# B&R Automation Studio project NAEUL004C00R13L518F00 (part 43)

#### Local.var
```iecst
(*2019-10-30*)
(**)
(*Local Action, State & Status*)
VAR
	eAct : eMagConv2ClpAction := MagConv2ClpActIdle;
	eStat : eMagConv2ClpAction := MagConv2ClpActIdle;
	eStatus : eFBStatus := Idle;
	udiStatus : UDINT := 0;
	sStatTxt : STRING[200] := '';
	a_sStatText : ARRAY[0..50] OF STRING[200] := ['Idling','Initializing','Initializing With Stop Then Clamper','Initializing With Clamper Then Stop','Entering Board','Entering Board With Stop Then Clamper','Entering Board With Clamper Then Stop','Pre-Exiting Board','Pre-Exiting Board With Clamper',2('Exiting Board'),2('Exiting Board With Clamper'),'Fix/Bottom Clamper Setting All Control','Fix/Bottom Clamper Resetting All Control','Fix/Bottom Clamper Setting Clamp','Fix/Bottom Clamper Setting Unclamp','Fix/Bottom Clamper Clamp','Fix/Bottom Clampler Unclamp','Remote/Top Clamper Setting All Control','Remote/Top Clamper Resetting All Control','Remote/Top Clamper Setting Clamp','Remote/Top Clamper Setting Unclamp','Remote/Top Clamper Clamp','Remote/Top Clampler Unclamp','Stopping','Stopping With Clamper','Turning On Motor Signal','Turning On Motor Direction','Turning Off Motor Signal','Turning Off Motor Direction','Turning On All Motor Output','Turning Off All Motor Output',18('')];
END_VAR
(**)
(*Local Alarm*)
VAR
	tyAlmData : tyAlmDat;
	a_tyAlmText : ARRAY[10000..10099] OF tyAlmTxt := [(sAlmText:='Magazine Detected But Not Present At Outlet Sensor (L - R) While Magazine Conveyor Initial',sRcyText:='Operation Interrupted By Undetected Magazine. Adjusting The Magazine Or Remove The Present Magazine To Resume Operation.'),(sAlmText:='Magazine Detected But Not Present At Outlet Sensor (R - L) While Magazine Conveyor Initial',sRcyText:='Operation Interrupted By Undetected Magazine. Adjusting The Magazine Or Remove The Present Magazine To Resume Operation.'),(sAlmText:='Clamper Clamp Sensor Off Time Out In Unclamp Check While Conveyor Initial With Clamper',sRcyText:='Sensor Timeout Expired Before Operation Completed. Sensor Operation Is Abnormal. Solve The Error To Resume Operation.'),(sAlmText:='Clamper Unclamp Sensor On Time Out In Unclamp Check While Conveyor Initial With Clamper',sRcyText:='Sensor Timeout Expired Before Operation Completed. Sensor Operation Is Abnormal. Solve The Error To Resume Operation.'),(sAlmText:='Clamper Unclamp Safety Sensor Error In Unclamp Check While Conveyor Initial With Clamper',sRcyText:='Safety System Has Been Triggered. All Operations Are Disable. Remove the Obstacle That Triggered The Safety Interlock To Resume Operation.'),(sAlmText:='Magazine Detected But Not Present At Outlet Sensor (L - R) While Conveyor Initial With Clamper',sRcyText:='Operation Interrupted By Undetected Magazine. Adjusting The Magazine Or Remove The Present Magazine To Resume Operation.'),(sAlmText:='Magazine Detected But Not Present At Outlet Sensor (R - L) While Conveyor Initial With Clamper',sRcyText:='Operation Interrupted By Undetected Magazine. Adjusting The Magazine Or Remove The Present Magazine To Resume Operation.'),(sAlmText:='Clamper Clamp Sensor On Time Out In Clamp Check While Conveyor Initial With Clamper',sRcyText:='Sensor Timeout Expired Before Operation Completed. Sensor Operation Is Abnormal. Solve The Error To Resume Operation.'),(sAlmText:='Clamper Unclamp Sensor Off Time Out In Clamp Check While Conveyor Initial With Clamper',sRcyText:='Sensor Timeout Expired Before Operation Completed. Sensor Operation Is Abnormal. Solve The Error To Resume Operation.'),(sAlmText:='Clamper Clamp Safety Sensor Error In Clamp Check While Conveyor Initial With Clamper',sRcyText:='Safety System Has Been Triggered. All Operations Are Disable. Remove the Obstacle That Triggered The Safety Interlock To Resume Operation.'),(sAlmText:='Clamper Clamp Sensor On Time Out In Clamp Check While Conveyor Enter With Clamper',sRcyText:='Sensor Timeout Expired Before Operation Completed. Sensor Operation Is Abnormal. Solve The Error To Resume Operation.'),(sAlmText:='Clamper Unclamp Sensor Off Time Out In Clamp Check While Conveyor Enter With Clamper',sRcyText:='Sensor Timeout Expired Before Operation Completed. Sensor Operation Is Abnormal. Solve The Error To Resume Operation.'),(sAlmText:='Clamper Clamp Safety Sensor Error In Clamp Check While Conveyor Enter With Clamper',sRcyText:='Safety System Has Been Triggered. All Operations Are Disable. Remove the Obstacle That Triggered The Safety Interlock To Resume Operation.'),(sAlmText:='Clamper Clamp Sensor Off Time Out In Unclamp Check While Conveyor Exit With Clamper',sRcyText:='Sensor Timeout Expired Before Operation Completed. Sensor Operation Is Abnormal. Solve The Error To Resume Operation.'),(sAlmText:='Clamper Unclamp Sensor On Time Out In Unclamp Check While Conveyor Exit With Clamper',sRcyText:='Sensor Timeout Expired Before Operation Completed. Sensor Operation Is Abnormal. Solve The Error To Resume Operation.'),(sAlmText:='Clamper Unclamp Safety Sensor Error In Unclamp Check While Conveyor Exit With Clamper',sRcyText:='Safety System Has Been Triggered. All Operations Are Disable. Remove the Obstacle That Triggered The Safety Interlock To Resume Operation.'),(sAlmText:='Clamper Clamp Sensor On Time Out In Clamp Check While Clamper Clamp',sRcyText:='Sensor Timeout Expired Before Operation Completed. Sensor Operation Is Abnormal. Solve The Error To Resume Operation.'),(sAlmText:='Clamper Unclamp Sensor Off Time Out In Clamp Check While Clamper Clamp',sRcyText:='Sensor Timeout Expired Before Operation Completed. Sensor Operation Is Abnormal. Solve The Error To Resume Operation.'),(sAlmText:='Clamper Clamp Safety Sensor Error In Clamp Check While Clamper Clamp',sRcyText:='Safety System Has Been Triggered. All Operations Are Disable. Remove the Obstacle That Triggered The Safety Interlock To Resume Operation.'),(sAlmText:='Clamper Clamp Sensor Off Time Out In Unclamp Check While Clamper Unclamp',sRcyText:='Sensor Timeout Expired Before Operation Completed. Sensor Operation Is Abnormal. Solve The Error To Resume Operation.'),(sAlmText:='Clamper Unclamp Sensor On Time Out In Unclamp Check While Clamper Unclamp',sRcyText:='Sensor Timeout Expired Before Operation Completed. Sensor Operation Is Abnormal. Solve The Error To Resume Operation.'),(sAlmText:='Clamper Unclamp Safety Sensor Error In Unclamp Check While Clamper Unclamp',sRcyText:='Safety System Has Been Triggered. All Operations Are Disable. Remove the Obstacle That Triggered The Safety Interlock To Resume Operation.'),(sAlmText:='Clamper Clamp Sensor Off Time Out In Unclamp Check While Stop With Clamper',sRcyText:='Sensor Timeout Expired Before Operation Completed. Sensor Operation Is Abnormal. Solve The Error To Resume Operation.'),(sAlmText:='Clamper Unclamp Sensor On Time Out In Unclamp Check While Stop With Clamper',sRcyText:='Sensor Timeout Expired Before Operation Completed. Sensor Operation Is Abnormal. Solve The Error To Resume Operation.'),(sAlmText:='Clamper Unclamp Safety Sensor Error In Unclamp Check While Stop With Clamper',sRcyText:='Safety System Has Been Triggered. All Operations Are Disable. Remove the Obstacle That Triggered The Safety Interlock To Resume Operation.'),(sAlmText:='Clamper Clamp Sensor Off Time Out In Unclamp Check While Conveyor Exit With Clamper',sRcyText:='Sensor Timeout Expired Before Operation Completed. Sensor Operation Is Abnormal. Solve The Error To Resume Operation.'),(sAlmText:='Clamper Unclamp Sensor On Time Out In Unclamp Check While Conveyor Exit With Clamper',sRcyText:='Sensor Timeout Expired Before Operation Completed. Sensor Operation Is Abnormal. Solve The Error To Resume Operation.'),(sAlmText:='Clamper Unclamp Safety Sensor Error In Unclamp Check While Conveyor Exit With Clamper',sRcyText:='Safety System Has Been Triggered. All Operations Are Disable. Remove the Obstacle That Triggered The Safety Interlock To Resume Operation.'),2((sAlmText:='Transfer In Time Out While Entering Magazine',sRcyText:='Timeout Expired Before Operation Completed. Transmission Abnormal. Remove the Obstacle (If Exists) To Resume Operation.')),(sAlmText:='Transfer Out Time Out While Exiting Magazine',sRcyText:='Timeout Expired Before Operation Completed. Transmission Abnormal. Remove the Obstacle (If Exists) To Resume Operation.'),(sAlmText:='Transfer Out Time Out While Conveyor Exit With Clamper',sRcyText:='Timeout Expired Before Operation Completed. Transmission Abnormal. Remove the Obstacle (If Exists) To Resume Operation.'),(sAlmText:='Transfer Out Time Out While Exiting Magazine',sRcyText:='Timeout Expired Before Operation Completed. Transmission Abnormal. Remove the Obstacle (If Exists) To Resume Operation.'),(sAlmText:='Transfer Out Time Out While Conveyor Exit With Clamper',sRcyText:='Timeout Expired Before Operation Completed. Transmission Abnormal. Remove the Obstacle (If Exists) To Resume Operation.'),(sAlmText:='Clamper Clamp Sensor On Time Out In Clamp Check While Conveyor Enter With Clamper',sRcyText:='Sensor Timeout Expired Before Operation Completed. Sensor Operation Is Abnormal. Solve The Error To Resume Operation.'),(sAlmText:='Clamper Unclamp Sensor Off Time Out In Clamp Check While Conveyor Enter With Clamper',sRcyText:='Sensor Timeout Expired Before Operation Completed. Sensor Operation Is Abnormal. Solve The Error To Resume Operation.'),(sAlmText:='Clamper Clamp Safety Sensor Error In Clamp Check While Conveyor Enter With Clamper',sRcyText:='Safety System Has Been Triggered. All Operations Are Disable. Remove the Obstacle That Triggered The Safety Interlock To Resume Operation.'),(sAlmText:='Transfer In Time Out While Entering Magazine',sRcyText:='Timeout Expired Before Operation Completed. Transmission Abnormal. Remove the Obstacle (If Exists) To Resume Operation.'),(sAlmText:='Clamper Clamp Sensor Off Time Out In Unclamp Check While Conveyor Initial With Clamper',sRcyText:='Sensor Timeout Expired Before Operation Completed. Sensor Operation Is Abnormal. Solve The Error To Resume Operation.'),(sAlmText:='Clamper Unclamp Sensor On Time Out In Unclamp Check While Conveyor Initial With Clamper',sRcyText:='Sensor Timeout Expired Before Operation Completed. Sensor Operation Is Abnormal. Solve The Error To Resume Operation.'),(sAlmText:='Clamper Unclamp Safety Sensor Error In Unclamp Check While Conveyor Initial With Clamper',sRcyText:='Safety System Has Been Triggered. All Operations Are Disable. Remove the Obstacle That Triggered The Safety Interlock To Resume Operation.'),(sAlmText:='Magazine Detected But Not Present At Outlet Sensor (L - R) While Conveyor Initial With Clamper',sRcyText:='Operation Interrupted By Undetected Magazine. Adjusting The Magazine Or Remove The Present Magazine To Resume Operation.'),(sAlmText:='Magazine Detected But Not Present At Outlet Sensor (R - L) While Conveyor Initial With Clamper',sRcyText:='Operation Interrupted By Undetected Magazine. Adjusting The Magazine Or Remove The Present Magazine To Resume Operation.'),(sAlmText:='Clamper Clamp Sensor On Time Out In Clamp Check While Conveyor Initial With Clamper',sRcyText:='Sensor Timeout Expired Before Operation Completed. Sensor Operation Is Abnormal. Solve The Error To Resume Operation.'),(sAlmText:='Clamper Unclamp Sensor Off Time Out In Clamp Check While Conveyor Initial With Clamper',sRcyText:='Sensor Timeout Expired Before Operation Completed. Sensor Operation Is Abnormal. Solve The Error To Resume Operation.'),(sAlmText:='Clamper Clamp Safety Sensor Error In Clamp Check While Conveyor Initial With Clamper',sRcyText:='Safety System Has Been Triggered. All Operations Are Disable. Remove the Obstacle That Triggered The Safety Interlock To Resume Operation.'),(sAlmText:='Magazine Not Detected While Pre-Exiting Magazine',sRcyText:='Operation Interrupted By Undetected Magazine. Adjusting The Magazine Or Remove The Present Magazine To Resume Operation.'),(sAlmText:='Magazine Width Check Sensor Deactivated',sRcyText:='Please Check the Magazine Width'),(sAlmText:='Saftey Sensor Is Deactivated To Clamp',sRcyText:='Please Check Safety Sensor'),51((0))];
END_VAR
(**)
(*Local Output*)
VAR
	bHvMag : BOOL := FALSE;
	bMtrSigOnOrLToR : BOOL := FALSE;
	bMtrDirOrRToL : BOOL := FALSE;
	bFixClprClampCtrl : BOOL;
	bRmtClprClampCtrl : BOOL;
	bClprTwoOutputControl : BOOL := FALSE;
END_VAR
(**)
(*Local Input*)
VAR
	udiRstErr : UDINT := 0;
	bPrep : BOOL := TRUE;
	bEn : BOOL := TRUE;
	bDis : BOOL := FALSE;
	bManual : BOOL := FALSE;
	bOnDirMod : BOOL := FALSE;
	diInitTm : DINT := 10000;
	tMtrOffDlyTm : TIME := T#0S;
	diTxInTimeOut : DINT := 10000;
	diTxOutTimeOut : DINT := 10000;
	eDirection : eConvDir := ConvDirLToR;
	bLeftSen : BOOL := FALSE;
	bRightSen : BOOL := FALSE;
	bFixClprClampSen : BOOL := FALSE;
	bFixClprUnclampSen : BOOL := FALSE;
	bFixClprClampSafetySen : BOOL := TRUE;
	bFixClprUnclampSafetySen : BOOL := TRUE;
	bRmtClprClampSen : BOOL := FALSE;
	bRmtClprUnclampSen : BOOL := FALSE;
	bRmtClprClampSafetySen : BOOL := TRUE;
	bRmtClprUnclampSafetySen : BOOL := TRUE;
	bWidthChkPrep : BOOL := TRUE;
	sProgNm : STRING[15] := 'MagConv2Clp';
	tClprClampTO : TIME := T#20s;
	tClprUnclampTO : TIME := T#20s;
	bNtSettingsLoadDone : BOOL := TRUE;
END_VAR
(**)
(*Local*)
VAR
	bRstErr : BOOL;
	udiRstErrOld : UDINT;
	bInitDone : BOOL;
	bInitialDone : BOOL;
	bReachEnd : BOOL;
	usiStep : USINT;
	usiSubStep : USINT;
	eStatOld : eMagConv2ClpAction := MagConv2ClpActIdle;
	fbInit : fbConvSenToSenTm;
	fbEnt : fbConvSenToSen;
	fbPreExit : fbConvSenToSenTm;
	fbExit : fbConvSenToSenOff;
	fbExit1 : fbConvSenToSenOff1;
	fbStop : fbConvMtrOff;
	fbFixClprClampChk : fbPneuExtRetSenExtChk;
	fbFixClprUnclampChk : fbPneuExtRetSenRetChk;
	fbRmtClprClampChk : fbPneuExtRetSenExtChk;
	fbFixClprDly : TON := (PT:=T#1s);
	fbRmtClprUnclampChk : fbPneuExtRetSenRetChk;
	fbClprDlyTm : TON;
	fbSmallLargeSenDlyTm : TON := (PT:=T#1S);
	fbWidthChk : TON := (PT:=T#30s);
	fbLeftSenDelayTm : TON := (PT:=T#1S);
	fbClpExtChkTm : TON := (PT:=T#200ms);
	udiModuleNum : UDINT := 1901;
END_VAR
```

#### Act_Alarm.st
```iecst
(** 2019-10-30 **)
ACTION Act_Alarm:
	//Reset Error
	IF (tylocalMagConv2Clp.Out.eStatus = Error) AND bRstErr THEN
		tylocalMagConv2Clp.In.eAct	:= MagConv2ClpActIdle;
		tylocalMagConv2Clp.Out.eStat	:= MagConv2ClpActIdle;
	END_IF

	IF tylocalMagConv2Clp.In.udiRstErr <> udiRstErrOld THEN
		bRstErr			:= TRUE;
		udiRstErrOld	:= tylocalMagConv2Clp.In.udiRstErr;
	ELSE
		bRstErr			:= FALSE;
	END_IF
	//Error
	IF EDGEPOS(tylocalMagConv2Clp.Out.eStatus = Error) THEN

		tylocalMagConv2Clp.Out.tyAlmData.sProgNm		:= tylocalMagConv2Clp.In.sProgNm;
		tylocalMagConv2Clp.Out.tyAlmData.udiCode		:= udiStatus;
		tylocalMagConv2Clp.Out.tyAlmData.eSeverity		:= AlmSeverityError;
		tylocalMagConv2Clp.Out.tyAlmData.udiRunTime	:= tylocalMagConv2Clp.Out.tyAlmData.udiRunTime + 1;
		tylocalMagConv2Clp.Out.tyAlmData.bAlm			:= TRUE;
		tylocalMagConv2Clp.Out.tyAlmData.udiModuleNum  := udiModuleNum;
		g_sMagConv2ClpProgNm		:= tylocalMagConv2Clp.In.sProgNm;
		tylocalMagConv2Clp.Out.sStatTxt	:= tylocalMagConv2Clp.Out.tyAlmData.sAlmMsg;

	ELSIF bRstErr AND (tylocalMagConv2Clp.Out.tyAlmData.udiCode <> 0) THEN

		tylocalMagConv2Clp.Out.tyAlmData.udiCode	:= 0;
		tylocalMagConv2Clp.Out.tyAlmData.eSeverity	:= AlmSeverityNA;
		tylocalMagConv2Clp.Out.tyAlmData.bAlm			:= FALSE;
		tylocalMagConv2Clp.Out.sStatTxt	:= a_sStatText[tylocalMagConv2Clp.Out.eStat];

	END_IF

END_ACTION
```

#### Act_InitGlobal.st
```iecst
(** 2019-10-30 **)
ACTION Act_InitGlobal:

	(* Always Change If Project Change *)

	//Pass Data To Link
	p_bLinkOpsRun ACCESS p_OpsRun;

	p_bLinkDISafetyRlySig ACCESS p_DISafetyRlySig;

	p_bLinkMagSmallSen ACCESS p_DIMagConvSmallMagSen2;
	p_bLinkMagLargeSen ACCESS p_DIMagConvLargeMagSen2;
	p_bLinkFixClprUnClampSen ACCESS p_DIMag2FixedUnclampRS;
	p_bLinkFixClprClampSen ACCESS p_DIMag2FixedClampRS; //Pneumatic Clamp RS
	p_bLinkFixClprMagDetectSen ACCESS p_DIMag2FixedClampSen; // Clamping Done Before Pneumatic Clamp Reed Switch for special Condition
	p_bLinkFixClprMagDetectSenPrep ACCESS p_NtParamProjFixClpMagDSenPrep; // Fixed Clamp Detect Sensor Prep before Clamp RS

	p_bLinkMagOpsStepMagFullExit ACCESS p_OpsMagConvUL2MagFullExit;
	p_bLinkDIMagEntSen ACCESS p_DIMagConvEntSen2;
	p_bLinkDO ACCESS p_DO;

	p_bLinkNtParamMagModelAutoVerify ACCESS p_NtParamProjMagAutoVerifyPrep;

	p_bWidthChkInterrupt ACCESS p_DICurtainSen;
	p_bWidthChkSen	ACCESS p_DIMagWidthChkSen;

	p_tyDISettings ACCESS p_NtParamDISettings;
	p_bLinkFixClprClampSen ACCESS ADR(bFixClprClampSen);//p_DIMag1FixedSideDetect;//p_DIMag1FixedClampRS; //initLocal at 1st

	//Pass Data To Internal Use
	p_udiRstErr ACCESS p_RstErrReset;
	p_bPrep ACCESS p_NtParamProjMag2ConvPrep;
	p_bManual ACCESS p_UIMnlMod;
	p_bOnDirMod ACCESS p_NtParamMagConv2OnDirMod;
	p_diInitTm ACCESS p_McParamMag2ConvRunTmOut;
	p_tMtrOffDlyTm ACCESS p_NtParamMagConv2MtrOffDlyTm;
	p_diTxInTimeOut ACCESS p_McParamMag2ConvRunTmOut;
	p_diTxOutTimeOut ACCESS p_McParamMag2ConvRunTmOut;
	p_eDirection ACCESS p_NtParamProjMagConvDir;
	p_sProgNm ACCESS p_NtParamMagConv2ProgNm;
	p_tClprClampTO ACCESS p_NtParamMagConv2ClprClampTO;
	p_tClprUnclampTO ACCESS p_NtParamMagConv2ClprUnclampTO;
//	p_bLeftSen ACCESS p_DIMagPresentSen2;
	p_bRightSen	ACCESS p_DIMagPresentSen2;

	p_bNtSettingsLoadDone ACCESS p_StartupNtSettingsLoadDone;

	(* Always Change If Project Change *)

END_ACTION
```

#### Act_Initial.st
```iecst
(** 2019-10-30 **)
ACTION Act_Initial:

	//Initial
	sStatTxt	:= a_sStatText[eStat];

	fbInit.bStartSen	:= TRUE;
	fbInit(bEn := FALSE);
	fbEnt.bStartSen		:= TRUE;
	fbEnt(bEn := FALSE);
	fbPreExit.bStartSen		:= TRUE;
	fbPreExit(bEn := FALSE);
	fbExit.bStartSen	:= TRUE;
	fbExit(bEn := FALSE);
	fbExit1.bStartSen		:= TRUE;
	fbExit1(bEn := FALSE);
	fbStop(bEn := FALSE);
	fbFixClprClampChk(bEn := FALSE);
	fbFixClprUnclampChk(bEn := FALSE);
	fbRmtClprClampChk(bEn := FALSE);
	fbRmtClprUnclampChk(bEn := FALSE);
	fbClprDlyTm(IN := FALSE);

END_ACTION
```

#### Act_InputConfig.st
```iecst
(** 2019-10-30 **)
ACTION Act_InputConfig:

	(* Always Change If Project Change *)

	//Pass Data To Link

	tylocalMagConv2Clp.In.bLinkDISafetyRlySig := g_tyDInput.bSafetyRlySig;

	tylocalMagConv2Clp.In.bLinkMagSmallSen := g_tyDInput.bMagConvSmallMagSen2;
	tylocalMagConv2Clp.In.bLinkMagLargeSen := g_tyDInput.bMagConvLargeMagSen2;
	tylocalMagConv2Clp.In.bLinkFixClprUnClampSen := g_tyDInput.bMag2FixedUnclampRS;
	//	tylocalMagConv2Clp.In.bLinkFixClprClampSen := g_tyDInput.bMag2FixedClampRS; // Pneumatic Clamp Reed Switch
	tylocalMagConv2Clp.In.bLinkFixClprMagDetectSen := g_tyDInput.bMag2FixedClampSen; // Clamping Done Before Pneumatic Clamp Reed Switch for special Condition
	tylocalMagConv2Clp.In.bLinkFixClprMagDetectSenPrep := g_tyNtParamCurr.bProjFixClpMagDSenPrep; // Fixed Clamp Detect Sensor Prep before Clamp RS

	tylocalMagConv2Clp.In.bLinkMagOpsStepMagFullExit := g_tyOpsMagConvUL2MagFullExit;
	tylocalMagConv2Clp.In.bLinkDIMagEntSen := g_tyDInput.bMagConvEntSen2;
	//	tylocalMagConv2Clp.In.bLinkDO := g_tyDO;

	tylocalMagConv2Clp.In.bWidthChkSen := g_tyNtParamCurr.bCurtainSenPrep;
	tylocalMagConv2Clp.In.bWidthChkInterrupt := g_tyDInput.bCurtainSen;

	tylocalMagConv2Clp.In.bLinkNtParamMagModelAutoVerify := g_tyNtParamCurr.bProjMagAutoVerifyPrep;
	//	tylocalMagConv2Clp.In.tyDISettings := g_tyNtParamCurr.tyDISettings;
	//	tylocalMagConv2Clp.In.bLinkFixClprClampSen ACCESS ADR(bFixClprClampSen);//tylocalMagConv2Clp.In.DIMag2FixedSideDetect;//tylocalMagConv2Clp.In.DIMag2FixedClampRS; //initLocal at 1st

	//Pass Data To Internal Use
	tylocalMagConv2Clp.In.udiRstErr := g_tyRstErrReset;
	tylocalMagConv2Clp.In.bPrep := g_tyNtParamCurr.bProjMag2ConvPrep;
	tylocalMagConv2Clp.In.bManual := g_tyUIMnlMod;
	tylocalMagConv2Clp.In.bOnDirMod := g_tyNtParamCurr.bMagConv2OnDirMod;
	tylocalMagConv2Clp.In.diInitTm := g_tyMcParamCurr.tMag2ConvRunTmOut;
	tylocalMagConv2Clp.In.tMtrOffDlyTm := g_tyNtParamCurr.tMagConv2MtrOffDlyTm;
	tylocalMagConv2Clp.In.diTxInTimeOut := g_tyMcParamCurr.tMag2ConvRunTmOut;
	tylocalMagConv2Clp.In.diTxOutTimeOut := g_tyMcParamCurr.tMag2ConvRunTmOut;
	tylocalMagConv2Clp.In.eDirection := g_tyNtParamCurr.bProjMagConvDir;
	tylocalMagConv2Clp.In.sProgNm := g_tyNtParamCurr.sMagConv2ProgNm;
	tylocalMagConv2Clp.In.tClprClampTO := g_tyNtParamCurr.tMagConv2ClprClampTO;
	tylocalMagConv2Clp.In.tClprUnclampTO := g_tyNtParamCurr.tMagConv2ClprUnclampTO;
	//	tylocalMagConv2Clp.In.bLeftSen := g_tyDInput.bMagPresentSen2;
	tylocalMagConv2Clp.In.bRightSen	:= g_tyDInput.bMagPresentSen2;

	(* Always Change If Project Change *)

	IF g_tyOps.bRun THEN
		tylocalMagConv2Clp.In.eAct := g_tyOpsMagConvUL2.eMagConv2ClpAct;
	ELSIF tylocalMagConv2Clp.In.bManual = TRUE THEN
		tylocalMagConv2Clp.In.eAct := g_tyUIOut.eMnlAct.eMagConv2Clp2Act;
	ELSE
		tylocalMagConv2Clp.In.eAct := eAct;
	END_IF
END_ACTION
```

#### Act_Link.st
```iecst
(** 2019-10-30 **)
ACTION Act_Link:

	IF p_bLinkDISafetyRlySig = FALSE THEN
		bFixClprClampCtrl	:= FALSE;
		bRmtClprClampCtrl	:= FALSE;
	END_IF

	p_bFixClprUnclampSen :=  p_bLinkFixClprUnClampSen;

	IF p_bLinkNtParamMagModelAutoVerify THEN
		fbSmallLargeSenDlyTm(IN:= p_bLinkMagSmallSen OR p_bLinkMagLargeSen);
		IF fbSmallLargeSenDlyTm.Q THEN
			p_bFixClprClampSen := TRUE;
		ELSE
			p_bFixClprClampSen := FALSE;
		END_IF
	ELSE
		IF p_bLinkFixClprMagDetectSenPrep THEN
			IF p_eAct = MagConv2ClpActFixClprUnclamp OR (p_eAct = MagConv2ClpActInitClpStop AND usiStep = 0) OR (p_eAct = MagConv2ClpActInitStopClp AND usiStep = 0)
				OR (p_eAct  = MagConv2ClpActPreExitClpr AND usiStep = 0) OR (p_eAct  = MagConv2ClpActExitClpr AND usiStep = 0)
				OR (p_eAct = MagConv2ClpActStopClpr) THEN

				p_bFixClprClampSen			:= NOT p_bLinkFixClprUnClampSen;
			ELSE
				p_bFixClprClampSen			:= p_bLinkFixClprMagDetectSen; //Treat as Clamping Sen Clamp RS for Special Case
			END_IF
			//p_bFixClprClampSafetySen	:= NOT p_bLinkFixClprClampSen; // If Clamping RS detects first, it will go to Error for safety check
		ELSE
			p_bFixClprClampSen := p_bLinkFixClprClampSen; //Normal Pneumatic Clamping RS.
		END_IF
	END_IF

	p_bRmtClprClampSen := p_bLinkDO.bMag2RemoteClampCtrl;
	p_bRmtClprUnclampSen := NOT p_bLinkDO.bMag2RemoteClampCtrl;
//	p_tMtrOffDlyTm	:= T#200ms;

	IF p_bLinkMagOpsStepMagFullExit THEN
		fbLeftSenDelayTm(IN:= TRUE, PT:=  T#3000ms);
	 	IF fbLeftSenDelayTm.Q THEN
				p_bLeftSen := p_bLinkDIMagEntSen;
		END_IF
	ELSE
		p_bLeftSen := p_bLinkDIMagEntSen;
		fbLeftSenDelayTm(IN:= FALSE);
	END_IF

	//Clamp Sensor chk time
	IF p_tyDISettings.diMag2FixedClampSen >0 THEN //fix side sensor used

		IF eStat = MagConv2ClpActInitStopClp AND usiStep = 3 OR
			eStat = MagConv2ClpActEntStopClp AND usiStep = 1 OR
			eStat = MagConv2ClpActFixClprClamp OR eStat = MagConv2ClpActFixClprUnclamp THEN //during clamp
			fbClpExtChkTm(IN:=TRUE);

			IF fbClpExtChkTm.Q THEN
				fbClpExtChkTm(IN:=FALSE);
				p_bLinkFixClprClampSen ACCESS p_DIMag2FixedClampSen;
			ELSE
				p_bLinkFixClprClampSen ACCESS ADR(bFixClprClampSen);
			END_IF
		ELSE
			fbClpExtChkTm(IN:=FALSE);
			p_bFixClprClampSen := FALSE;
		END_IF
	ELSE //standard 2 RS
		p_bLinkFixClprClampSen ACCESS p_DIMag2FixedClampRS;
	END_IF

END_ACTION
```

#### Act_LinkAction.st
```iecst
(** 2019-10-30 **)
ACTION Act_LinkAction:

	IF p_bLinkOpsRun = TRUE THEN
		p_eAct ACCESS p_OpsMagConvUL2MagConv2ClpAct;
	ELSIF p_bManual = TRUE THEN
		p_eAct ACCESS p_UIMagConv2Clp2Act;
	ELSE
		p_eAct ACCESS ADR(eAct);
	END_IF

END_ACTION
```

#### Act_OutputConfig.st
```iecst
ACTION Act_OutputConfig:
	// Output: Assign To Global For Independent Package Usage

	g_tyPneuMag2AWEngage := tylocalMagConv2Clp.Out; // Change the Global Naming According to the Physical Hardware Module

END_ACTION
```

#### Act_RstErr.st
```iecst
(** 2019-10-30 **)
ACTION Act_RstErr:

	IF p_udiRstErr <> udiRstErrOld THEN
		bRstErr			:= TRUE;
		udiRstErrOld	:= p_udiRstErr;
	ELSE
		bRstErr			:= FALSE;
	END_IF

END_ACTION
```

#### Cyclic.st
```iecst
(** 2019-10-30 **)
PROGRAM _CYCLIC

	IF bInitialDone = FALSE THEN
		IF g_tyStartUp.bNtSettingsLoadDone = TRUE  THEN
			bInitialDone	:= TRUE;
			Act_Initial;
		END_IF
	ELSE
		Act_InputConfig;
		IF (tylocalMagConv2Clp.In.bPrep = TRUE) AND (tylocalMagConv2Clp.In.bEn = TRUE) AND (tylocalMagConv2Clp.In.bDis = FALSE) THEN
			Act_Link;
			Act_Main;
		ELSE
			IF tylocalMagConv2Clp.Out.eStat <> MagConv2ClpActIdle THEN
				tylocalMagConv2Clp.Out.eStatus	:= Done;
			ELSE
				tylocalMagConv2Clp.Out.eStatus	:= Idle;
			END_IF
		END_IF
		Act_OutputConfig;
		Act_Alarm;
	END_IF

END_PROGRAM
```

#### Init.st
```iecst
(** 2019-10-30 **)
PROGRAM _INIT

	(* Always Change If Project Change *)

	//Pass Address To Global Address For External Use
	//Action, State & Status
	p_MagConv2Clp2Stat		:= ADR(eStat);
	p_MagConv2Clp2Status	:= ADR(eStatus);
	p_MagConv2Clp2StatTxt	:= ADR(sStatTxt);

	//Alarm
	p_MagConv2Clp2AlmData	:= ADR(tyAlmData);

	//Output
	p_MagConv2Clp2HvMag				:= ADR(bHvMag);
	p_MagConv2Clp2MtrSigOnOrLToR	:= ADR(bMtrSigOnOrLToR);
	p_MagConv2Clp2MtrDirOrRToL		:= ADR(bMtrDirOrRToL);

	p_MagConv2Clp2FixClprClampCtrl	:= ADR(bFixClprClampCtrl);
	p_MagConv2Clp2RmtClprClampCtrl	:= ADR(bRmtClprClampCtrl);
	p_MagConv2Clp2ClprTwoOutputCtrl	:= ADR(bClprTwoOutputControl);

	(* Always Change If Project Change *)

END_PROGRAM
```

### Program Logical/MagConv_LiftnTrav/MagConv2Clp3 (IEC, version 1.00.0) - 1.00.0 - NtConv v5.00.0 , NtPneu v5.00.0

#### Init.st - Change By Project
```iecst
(** 2019-10-30 **)
PROGRAM _INIT

	(* Always Change If Project Change *)

	//Pass Address To Global Address For External Use
	//Action, State & Status
	p_MagConv2Clp3Stat				:= ADR(eStat);
	p_MagConv2Clp3Status			:= ADR(eStatus);
	p_MagConv2Clp3StatTxt			:= ADR(sStatTxt);

	//Alarm
	p_MagConv2Clp3AlmData			:= ADR(tyAlmData);

	//Output
	p_MagConv2Clp3HvMag				:= ADR(bHvMag);
	p_MagConv2Clp3MtrSigOnOrLToR	:= ADR(bMtrSigOnOrLToR);
	p_MagConv2Clp3MtrDirOrRToL		:= ADR(bMtrDirOrRToL);

	p_MagConv2Clp3FixClprClampCtrl	:= ADR(bFixClprClampCtrl);
	p_MagConv2Clp3RmtClprClampCtrl	:= ADR(bRmtClprClampCtrl);
	p_MagConv2Clp3ClprTwoOutputCtrl	:= ADR(bClprTwoOutputControl);

	(* Always Change If Project Change *)

END_PROGRAM
```

#### Act_InitGlobal.st - Change By Project
```iecst
(** 2019-10-30 **)
ACTION Act_InitGlobal:

	(* Always Change If Project Change *)

	//Pass Data To Link
	p_bLinkOpsRun ACCESS p_OpsRun;

	p_bLinkDISafetyRlySig ACCESS p_DISafetyRlySig;

	p_bLinkMagSmallSen ACCESS p_DIMagConvSmallMagSen3;
	p_bLinkMagLargeSen ACCESS p_DIMagConvLargeMagSen3;
	p_bLinkFixClprUnClampSen ACCESS p_DIMag3FixedUnclampRS;
	p_bLinkFixClprClampSen ACCESS p_DIMag3FixedClampRS; //Pneumatic Clamp RS
	p_bLinkFixClprMagDetectSen ACCESS p_DIMag3FixedClampSen; // Clamping Done Before Pneumatic Clamp Reed Switch for special Condition
	p_bLinkFixClprMagDetectSenPrep ACCESS p_NtParamProjFixClpMagDSenPrep; // Fixed Clamp Detect Sensor Prep before Clamp RS

	p_bLinkMagOpsStepMagFullExit ACCESS p_OpsMagConvUL3MagFullExit;
	p_bLinkDIMagEntSen ACCESS p_DIMagConvEntSen3;
	p_bLinkDO ACCESS p_DO;

	p_bLinkNtParamMagModelAutoVerify ACCESS p_NtParamProjMagAutoVerifyPrep;

	p_bWidthChkInterrupt ACCESS p_DICurtainSen;
	p_bWidthChkSen	ACCESS p_DIMagWidthChkSen;

	p_tyDISettings ACCESS p_NtParamDISettings;
	p_bLinkFixClprClampSen ACCESS ADR(bFixClprClampSen);//p_DIMag1FixedSideDetect;//p_DIMag1FixedClampRS; //initLocal at 1st

	//Pass Data To Internal Use
	p_udiRstErr ACCESS p_RstErrReset;
	p_bPrep ACCESS p_NtParamProjMag3ConvPrep;
	p_bManual ACCESS p_UIMnlMod;
	p_bOnDirMod ACCESS p_NtParamMagConv3OnDirMod;
	p_diInitTm ACCESS p_McParamMag3ConvRunTmOut;
	p_tMtrOffDlyTm ACCESS p_NtParamMagConv3MtrOffDlyTm;
	p_diTxInTimeOut ACCESS p_McParamMag3ConvRunTmOut;
	p_diTxOutTimeOut ACCESS p_McParamMag3ConvRunTmOut;
	p_eDirection ACCESS p_NtParamProjMagConvDir;
	p_sProgNm ACCESS p_NtParamMagConv3ProgNm;
	p_tClprClampTO ACCESS p_NtParamMagConv3ClprClampTO;
	p_tClprUnclampTO ACCESS p_NtParamMagConv3ClprUnclampTO;
//	p_bLeftSen ACCESS p_DIMagPresentSen3;
	p_bRightSen	ACCESS p_DIMagPresentSen3;

	p_bNtSettingsLoadDone ACCESS p_StartupNtSettingsLoadDone;

	(* Always Change If Project Change *)

END_ACTION
```

#### Act_LinkAction.st - Change By Project
```iecst
(** 2019-10-30 **)
ACTION Act_LinkAction:

	IF p_bLinkOpsRun = TRUE THEN
		p_eAct ACCESS p_OpsMagConvUL3MagConv2ClpAct;
	ELSIF p_bManual = TRUE THEN
		p_eAct ACCESS p_UIMagConv2Clp3Act;
	ELSE
		p_eAct ACCESS ADR(eAct);
	END_IF

END_ACTION
```

#### Act_Link.st - Change By Project
```iecst
(** 2019-10-30 **)
ACTION Act_Link:

	IF p_bLinkDISafetyRlySig = FALSE THEN
		bFixClprClampCtrl	:= FALSE;
		bRmtClprClampCtrl	:= FALSE;
	END_IF

	p_bFixClprUnclampSen :=  p_bLinkFixClprUnClampSen;

	IF p_bLinkNtParamMagModelAutoVerify THEN
		fbSmallLargeSenDlyTm(IN:= p_bLinkMagSmallSen OR p_bLinkMagLargeSen);
		IF fbSmallLargeSenDlyTm.Q THEN
			p_bFixClprClampSen := TRUE;
		ELSE
			p_bFixClprClampSen := FALSE;
		END_IF
	ELSE
		IF p_bLinkFixClprMagDetectSenPrep THEN
			IF p_eAct = MagConv2ClpActFixClprUnclamp OR (p_eAct = MagConv2ClpActInitClpStop AND usiStep = 0) OR (p_eAct = MagConv2ClpActInitStopClp AND usiStep = 0)
				OR (p_eAct  = MagConv2ClpActPreExitClpr AND usiStep = 0) OR (p_eAct  = MagConv2ClpActExitClpr AND usiStep = 0)
				OR (p_eAct = MagConv2ClpActStopClpr) THEN

				p_bFixClprClampSen			:= NOT p_bLinkFixClprUnClampSen;
			ELSE
				p_bFixClprClampSen			:= p_bLinkFixClprMagDetectSen; //Treat as Clamping Sen Clamp RS for Special Case
			END_IF
			//p_bFixClprClampSafetySen	:= NOT p_bLinkFixClprClampSen; // If Clamping RS detects first, it will go to Error for safety check
		ELSE
			p_bFixClprClampSen := p_bLinkFixClprClampSen; //Normal Pneumatic Clamping RS.
		END_IF
	END_IF

	p_bRmtClprClampSen := p_bLinkDO.bMag3RemoteClampCtrl;
	p_bRmtClprUnclampSen := NOT p_bLinkDO.bMag3RemoteClampCtrl;
//	p_tMtrOffDlyTm	:= T#200ms;

	IF p_bLinkMagOpsStepMagFullExit THEN
		fbLeftSenDelayTm(IN:= TRUE, PT:=  T#3000ms);
	 	IF fbLeftSenDelayTm.Q THEN
				p_bLeftSen := p_bLinkDIMagEntSen;
		END_IF
	ELSE
		p_bLeftSen := p_bLinkDIMagEntSen;
		fbLeftSenDelayTm(IN:= FALSE);
	END_IF

	//Clamp Sensor chk time
	IF p_tyDISettings.diMag3FixedClampSen >0 THEN //fix side sensor used

		IF eStat = MagConv2ClpActInitStopClp AND usiStep = 3 OR
			eStat = MagConv2ClpActEntStopClp AND usiStep = 1 OR
			eStat = MagConv2ClpActFixClprClamp OR eStat = MagConv2ClpActFixClprUnclamp THEN //during clamp
			fbClpExtChkTm(IN:=TRUE);

			IF fbClpExtChkTm.Q THEN
				fbClpExtChkTm(IN:=FALSE);
				p_bLinkFixClprClampSen ACCESS p_DIMag3FixedClampSen;
			ELSE
				p_bLinkFixClprClampSen ACCESS ADR(bFixClprClampSen);
			END_IF
		ELSE
			fbClpExtChkTm(IN:=FALSE);
			p_bFixClprClampSen := FALSE;
		END_IF
	ELSE //standard 2 RS
		p_bLinkFixClprClampSen ACCESS p_DIMag3FixedClampRS;
	END_IF

END_ACTION
```

#### Act_LinkEn.st - Change By Project
```iecst
(** 2019-10-30 **)
ACTION Act_LinkEn:

	//Link bPrep, bEn & bDis

END_ACTION
```

#### Cyclic.st - Do Not Change!!!
```iecst
(** 2019-10-30 **)
PROGRAM _CYCLIC

	IF bInitialDone = FALSE THEN
		IF g_tyStartUp.bNtSettingsLoadDone = TRUE  THEN
			bInitialDone	:= TRUE;
			Act_Initial;
		END_IF
	ELSE
		Act_InputConfig;
		IF (p_bPrep = TRUE) AND (p_bEn = TRUE) AND (p_bDis = FALSE) THEN
			Act_Link;
			Act_Main;
		ELSE
			IF eStat <> MagConv2ClpActIdle THEN
				eStatus	:= Done;
			ELSE
				eStatus	:= Idle;
			END_IF
		END_IF
		Act_OutputConfig;
		Act_Alarm;
	END_IF

END_PROGRAM
```

#### Act_InitLocal.st - Do Not Change!!!
```iecst
(** 2019-10-30 **)
ACTION Act_InitLocal:

	//Input Reference Link To Local Variable
	p_eAct ACCESS ADR(eAct);
	p_udiRstErr ACCESS ADR(udiRstErr);
	p_bPrep ACCESS ADR(bPrep);
	p_bEn ACCESS ADR(bEn);
	p_bDis ACCESS ADR(bDis);

	p_bManual ACCESS ADR(bManual);
	p_bOnDirMod ACCESS ADR(bOnDirMod);
	p_diInitTm ACCESS ADR(diInitTm);
	p_tMtrOffDlyTm ACCESS ADR(tMtrOffDlyTm);
	p_diTxInTimeOut ACCESS ADR(diTxInTimeOut);
	p_diTxOutTimeOut ACCESS ADR(diTxOutTimeOut);
	p_eDirection ACCESS ADR(eDirection);
	p_sProgNm ACCESS ADR(sProgNm);
	p_tClprClampTO ACCESS ADR(tClprClampTO);
	p_tClprUnclampTO ACCESS ADR(tClprUnclampTO);
	p_bNtSettingsLoadDone ACCESS ADR(bNtSettingsLoadDone);
	p_bLeftSen ACCESS ADR(bLeftSen);
	p_bRightSen ACCESS ADR(bRightSen);
	p_bFixClprClampSen ACCESS ADR(bFixClprClampSen);
	p_bFixClprUnclampSen ACCESS ADR(bFixClprUnclampSen);
	p_bFixClprClampSafetySen ACCESS ADR(bFixClprClampSafetySen);
	p_bFixClprUnclampSafetySen ACCESS ADR(bFixClprUnclampSafetySen);
	p_bRmtClprClampSen ACCESS ADR(bRmtClprClampSen);
	p_bRmtClprUnclampSen ACCESS ADR(bRmtClprUnclampSen);
	p_bRmtClprClampSafetySen ACCESS ADR(bRmtClprClampSafetySen);
	p_bRmtClprUnclampSafetySen ACCESS ADR(bRmtClprUnclampSafetySen);
	p_bWidthChkSenPrep ACCESS ADR (bWidthChkPrep);

END_ACTION
```

#### Act_Initial.st - Do Not Change!!!
```iecst
(** 2019-10-30 **)
ACTION Act_Initial:

	//Initial
	sStatTxt	:= a_sStatText[eStat];

	fbInit.bOnDirMod	:= p_bOnDirMod;
	fbInit.bStartSen	:= TRUE;
	fbInit.tMtrOffDlyTm	:= p_tMtrOffDlyTm;
	fbInit(bEn := FALSE);

	fbEnt.bOnDirMod		:= p_bOnDirMod;
	fbEnt.bStartSen		:= TRUE;
	fbEnt.tMtrOffDlyTm	:= p_tMtrOffDlyTm;
	fbEnt(bEn := FALSE);

	fbPreExit.bOnDirMod		:= p_bOnDirMod;
	fbPreExit.bStartSen		:= TRUE;
	fbPreExit.tMtrOffDlyTm	:= p_tMtrOffDlyTm;
	fbPreExit(bEn := FALSE);

	fbExit.bOnDirMod	:= p_bOnDirMod;
	fbExit.bStartSen	:= TRUE;
	fbExit.tMtrOffDlyTm	:= p_tMtrOffDlyTm;
	fbExit(bEn := FALSE);

	fbExit1.bOnDirMod		:= p_bOnDirMod;
	fbExit1.bStartSen		:= TRUE;
	fbExit1.tMtrOffDlyTm	:= p_tMtrOffDlyTm;
	fbExit1(bEn := FALSE);

	fbStop(bEn := FALSE);

	fbFixClprClampChk.tTimeOut	:= p_tClprClampTO;
	fbFixClprClampChk(bEn := FALSE);

	fbFixClprUnclampChk.tTimeOut	:= p_tClprUnclampTO;
	fbFixClprUnclampChk(bEn := FALSE);

	fbRmtClprClampChk.tTimeOut	:= p_tClprClampTO;
	fbRmtClprClampChk(bEn := FALSE);

	fbRmtClprUnclampChk.tTimeOut	:= p_tClprUnclampTO;
	fbRmtClprUnclampChk(bEn := FALSE);

	//Added
	fbFixClprUnclampChk1.tTimeOut := p_tClprClampTO;
	fbFixClprUnclampChk(bEn := FALSE);
	fbRmtClprUnclampChk1.tTimeOut := p_tClprUnclampTO;
	fbRmtClprUnclampChk1(bEn := FALSE);

	fbClprDlyTm.PT	:= p_tMtrOffDlyTm / 2;
	fbClprDlyTm(IN := FALSE);

END_ACTION
```
